Staubli VAL3: notGrip.pgx

program notGrip()
begin
  if switchGripper==true
    switchGripper=false
  else
  endIf
end
